Fanuc KAREL source: kb00144.KL

-- PROVISIONAL review KL for V1013-1; original PC SHA256 296153d44b16390919fb73d51fcd94ecc7aeec0768b999b1f7718a3967db950a
-- Incomplete behavior may be omitted. Consult companion uncertainty JSON. Do not deploy.
PROGRAM KB00144
%NOLOCKGROUP
BEGIN
  -- UNRESOLVED_PC offsets 5-14; opcodes 3F,75
  -- UNRESOLVED_PC offsets 19-26; opcodes 9D,23
  -- UNRESOLVED_PC offsets 31-38; opcodes 9D,23
  -- UNRESOLVED_PC offsets 43-50; opcodes 9D,23
  -- UNRESOLVED_PC offsets 55-62; opcodes 9D,23
  -- UNRESOLVED_PC offsets 67-109; opcodes 27,22,2A,22,22,22,22,22,31
  -- UNRESOLVED_PC offsets 114-118; opcodes 7F
END KB00144
